(*********************************** G.D S.p.A. - Technical Department ***********************************
============= PROGRAM INFO ============
FOLDER:             TBD
MACHINES INVOLVED:  TBD 

============= DESCRIPTION =============

============= REVISIONS ===============
Date		Version	 	Author      	Description             
----------	-------		------------  	--------------------------------------------
2019/04/24 	0000.00	 	M.Grasso		Creation of the PRG

**********************************************************************************************************)
(*$R 
	process_ref:= prc; 
$*)
PROGRAM csp_case_main_safety_drives_SD2200
VAR
	prc:					process;
	prc_path:				STRING;	

	sig:												safety_integrated_group;
	chA_smes_sis:										safety_integrated_series;
	chB_smes_sis:										safety_integrated_series;
	safety_integrated_series_close_dvr_chA: 			BOOL;
	safety_integrated_series_close_dvr_chB: 			BOOL;

	shutdown_chA AT %Q* 								:BOOL := TRUE;
	shutdown_chB AT %Q* 								:BOOL := TRUE;
END_VAR

_read_var_input();

_objects_manager();

IF NOT objects_running()
THEN
	RETURN;	
END_IF

_read_process_image();

_mode_manager();

//safety_integrated_series_close(chA_smes_sis);
//safety_integrated_series_close(chB_smes_sis);

IF  safety_integrated_series_get_mode (chA_smes_sis) = MODE_ABSENT
	OR
	safety_integrated_series_get_mode(chA_smes_sis) = MODE_INACTIVE
	THEN
		shutdown_chA := TRUE;
	ELSE
		shutdown_chA := FALSE;
END_IF

IF  safety_integrated_series_get_mode (chB_smes_sis) = MODE_ABSENT
	OR
	safety_integrated_series_get_mode(chB_smes_sis) = MODE_INACTIVE
	THEN
		shutdown_chB := TRUE;
	ELSE
		shutdown_chB := FALSE;
END_IF

CASE process_get_mode(prc) OF
	MODE_ABSENT,
	MODE_INACTIVE:
		RETURN;
	MODE_TEST:
		;
END_CASE

_set_runtime_properties();

(********************************* BODY *********************************)
IF NOT safety_integrated_group_is_running(sig)
		THEN
			safety_integrated_group_run(sig);
END_IF
safety_integrated_series_close(chA_smes_sis);
safety_integrated_series_close(chB_smes_sis);
safety_integrated_series_close_dvr_chA := safety_integrated_series_is_safely_closed(chA_smes_sis);
safety_integrated_series_close_dvr_chB := safety_integrated_series_is_safely_closed(chB_smes_sis);
(************************************************************************)

_handle_messages();

_write_output();

ACTION _handle_messages:
;
END_ACTION

ACTION _handle_process_test:
;
END_ACTION

ACTION _mode_manager:
IF process_mode_req_is_pending(prc)
THEN
    process_apply_mode_req_first_step(prc);
    CASE process_get_mode(prc) OF
        MODE_TO_ABSENT:
			;
        MODE_TO_INACTIVE:
			;
        MODE_TO_TEST:
			;
        MODE_TO_OPERATIONAL:
			;
    END_CASE
    process_apply_mode_req_second_step(prc);
END_IF
END_ACTION

ACTION _objects_manager:
IF objects_initialization()
THEN
	sub_process_init(
		object_name					:= 'csp_case_main_safety_drives_SD2200.prc', 
		process						:= csp_case_main_safety_drives.prc, 
		CONVERSION_this				:= prc);
		
	prc_path 						:= process_get_path(prc);

	safety_integrated_group_init(
        object_name				:=	CONCAT(prc_path, '_sig'), 
		controller				:=	csp_case_main_safety_interface.SPLC5000_sic,
        process					:=	prc,
        CONVERSION_this			:=	sig);

	(* Channel A SMES series *)
	safety_integrated_series_init(
		object_name				:=	CONCAT(prc_path, '_chA_smes_sis'), 
		_type					:=	SAFETY_INTEGRATED_SERIES_TYPE_NO_RESET,
		discrepancy_active		:=	TRUE,
		forced_open_active		:=	TRUE,
		process					:=	prc,
		CONVERSION_this			:=	chA_smes_sis);

	safety_integrated_series_add_safety_integrated_group(
		group					:=	sig,
		CONVERSION_this			:=	chA_smes_sis);

	safety_integrated_series_add_safety_integrated_series(
		series_active			:=	TRUE,
		series_polarity_direct	:=	TRUE,
		contact					:=	csp_case_main_safety_drives_commonConfiguration.rack_smes_sis, (*Marco : To be checked*)
		CONVERSION_this			:=	chA_smes_sis);
		
	(* Channel B SMES series *)
	safety_integrated_series_init(
		object_name				:=	CONCAT(prc_path, '_chB_smes_sis'), 
		_type					:=	SAFETY_INTEGRATED_SERIES_TYPE_NO_RESET,
		discrepancy_active		:=	TRUE,
		forced_open_active		:=	TRUE,
		process					:=	prc,
		CONVERSION_this			:=	chB_smes_sis);

	safety_integrated_series_add_safety_integrated_group(
		group					:=	sig,
		CONVERSION_this			:=	chB_smes_sis);
		
	safety_integrated_series_add_safety_integrated_series(
		series_active			:=	TRUE,
		series_polarity_direct	:=	TRUE,
		contact					:=	csp_case_main_safety_drives_commonConfiguration.rack_smes_sis, (*Marco : To be checked*)
		CONVERSION_this			:=	chB_smes_sis);
		
END_IF

IF objects_running()
THEN
	process_cycle(prc);
  	safety_integrated_group_cycle(sig);
	safety_integrated_series_cycle(chA_smes_sis);
	safety_integrated_series_cycle(chB_smes_sis);
END_IF
END_ACTION

ACTION _read_process_image:
;
END_ACTION

ACTION _read_var_input:
;
END_ACTION

ACTION _set_runtime_properties:
;
END_ACTION

ACTION _write_output:
;
END_ACTION

END_PROGRAM

(* stored: Version 1.1.0.1, ProductVersion 3.1.4024.3
   POU csp_case_main_safety_drives_SD2200: Id {abebf500-694f-4969-a168-f9b1aa494e0c}, SpecialFunc None
   Action _handle_messages: Id {c4b989a6-500d-4a8c-8bca-7d7b98530bc7}
   Action _handle_process_test: Id {fba19549-b5cf-407a-8145-65dceb24747f}
   Action _mode_manager: Id {5bc78058-9b68-405e-a2f0-282c43100b59}
   Action _objects_manager: Id {5edf1582-6b47-45f8-a758-eca292c713ad}
   Action _read_process_image: Id {0cdf0fc4-63f1-45d5-8894-875b4b37a42e}
   Action _read_var_input: Id {1ccb26b3-10ea-4144-9a56-25051e76171a}
   Action _set_runtime_properties: Id {e9f64353-4d63-44a5-9238-d80c21ba2d25}
   Action _write_output: Id {a3f3b656-835f-4b33-840e-d61774efef19} *)
